FUNCTION_BLOCK EL1804
VAR
	_io : EL1xx4_Data;
	{attribute addProperty Name "WcState"}
	_wcState : WcStateInputToggle;
	{attribute addProperty Name "Info data"}
	_infoData : InfoDataBase;
END_VAR

PROPERTY IO : REFERENCE TO EL1xx4_Data
GET
IO REF= _io;
END_GET
END_PROPERTY

PROPERTY WcState : REFERENCE TO WcStateInputToggle
GET
WcState REF= _wcState;
END_GET
END_PROPERTY

END_FUNCTION_BLOCK

(* stored: Version 1.1.0.1, ProductVersion 3.1.4024.9
   POU EL1804: Id {a2455aa2-4716-0612-2dfb-18fca29cab00}, SpecialFunc None
   Property IO: Id {73c54489-bab9-0785-345f-6e8467db7aad}
   Get Get: Id {d0fe9f00-f20a-00d1-2053-a84d4fd66578}
   Property WcState: Id {70bb12bd-fdb6-06e4-0455-3c3bd865815f}
   Get Get: Id {815014b1-69c1-0505-1464-9f6d94199e63} *)
